FUNCTION_BLOCK RequestManager (* Basic Function Block Type *)
  (* Standard: 61499-2 *)
  (* Version 0.0, 9/24/2026, macie, Schneider Electric, Template *)
  PACKAGE Main;
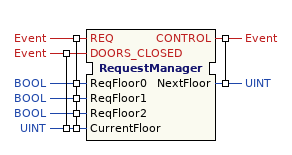
  EVENT_INPUT
    REQ WITH ReqFloor0, ReqFloor1, ReqFloor2, CurrentFloor; (* Normal Execution Request *)
    DOORS_CLOSED WITH CurrentFloor;
  END_EVENT
  EVENT_OUTPUT
    CONTROL WITH NextFloor; (* Initialization Confirm *)
  END_EVENT
  VAR_INPUT
    ReqFloor0 : BOOL;
    ReqFloor1 : BOOL;
    ReqFloor2 : BOOL;
    CurrentFloor : UINT;
  END_VAR
  VAR_OUTPUT
    NextFloor : UINT := 2; (* Output event qualifier *)
  END_VAR
  VAR
    Queue : ARRAY [0..2] OF UINT := [3(0)];
    MaxPriority : UINT;
    FloorPriority : UINT;
    QueueActive : BOOL := FALSE;
  END_VAR
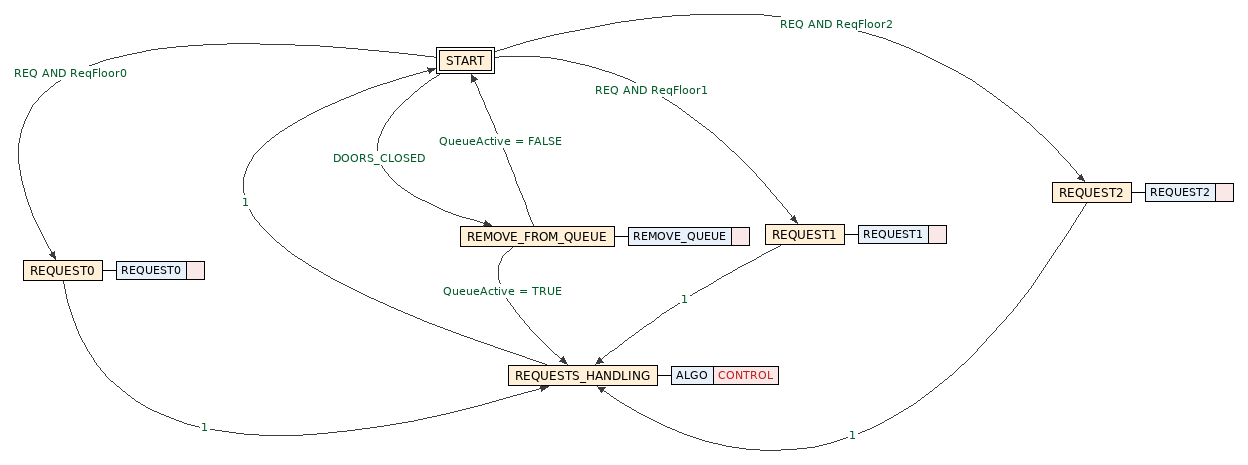
  EC_STATES
    START; (* Initial State *)
    REMOVE_FROM_QUEUE : REMOVE_QUEUE;
    REQUEST0 : REQUEST0;
    REQUEST1 : REQUEST1;
    REQUEST2 : REQUEST2;
    REQUESTS_HANDLING : ALGO -> CONTROL;
  END_STATES
  EC_TRANSITIONS
    START TO REMOVE_FROM_QUEUE := DOORS_CLOSED;
    START TO REQUEST0 := REQ AND ReqFloor0;
    REQUEST0 TO REQUESTS_HANDLING := 1;
    REQUEST1 TO REQUESTS_HANDLING := 1;
    REQUEST2 TO REQUESTS_HANDLING := 1;
    START TO REQUEST1 := REQ AND ReqFloor1;
    START TO REQUEST2 := REQ AND ReqFloor2;
    REMOVE_FROM_QUEUE TO START := QueueActive = FALSE;
    REMOVE_FROM_QUEUE TO REQUESTS_HANDLING := QueueActive = TRUE;
    REQUESTS_HANDLING TO START := 1;
  END_TRANSITIONS
  ALGORITHM ALGO IN ST: (* Initialization algorithm *)
;

NextFloor := CurrentFloor;
QueueActive := TRUE;
IF Queue[0] = 1 THEN
    IF CurrentFloor = 2 AND (Queue[1] > 0) THEN
        NextFloor := 1; (* Przystanek na 1 *)
    ELSE
        NextFloor := 0;
    END_IF;

ELSIF Queue[1] = 1 THEN
    NextFloor := 1;

ELSIF Queue[2] = 1 THEN
    IF CurrentFloor = 0 AND (Queue[1] > 0) THEN
        NextFloor := 1; (* Przystanek na 1 *)
    ELSE
        NextFloor := 2;
    END_IF;
END_IF;


(* --- 4. AKTUALIZACJA FLAGI AKTYWNOŚCI KOLEJKI --- *)
(* Ponownie przeliczamy priorytet, bo mógł zostać wyzerowany w Sekcji 2 *)
MaxPriority := MAX(Queue[0], MAX(Queue[1], Queue[2]));

IF FloorPriority = 0 THEN
    QueueActive := FALSE;
ELSE
    QueueActive := TRUE;
END_IF;
  END_ALGORITHM
  ALGORITHM REMOVE_QUEUE IN ST:
;
MaxPriority := MAX(Queue[0], MAX(Queue[1], Queue[2]));
IF MaxPriority > 0 THEN

	FloorPriority := Queue[CurrentFloor];
	Queue[CurrentFloor] := 0;


	IF Queue[0] > FloorPriority THEN Queue[0] := Queue[0] - 1; END_IF;
	IF Queue[1] > FloorPriority THEN Queue[1] := Queue[1] - 1; END_IF;
	IF Queue[2] > FloorPriority THEN Queue[2] := Queue[2] - 1; END_IF;
END_IF;

(*Updated value*)
MaxPriority := MAX(Queue[0], MAX(Queue[1], Queue[2]));

IF MaxPriority > 0 THEN
	QueueActive := TRUE;
ELSE
	QueueActive := FALSE;
END_IF;
  END_ALGORITHM
  ALGORITHM REQUEST0 IN ST:
;
MaxPriority := MAX(Queue[0], MAX(Queue[1], Queue[2]));

IF ReqFloor0 AND (Queue[0] = 0) THEN
    MaxPriority := MaxPriority + 1;
    Queue[0] := MaxPriority;
END_IF;
  END_ALGORITHM
  ALGORITHM REQUEST1 IN ST:
;
MaxPriority := MAX(Queue[0], MAX(Queue[1], Queue[2]));

IF ReqFloor1 AND (Queue[1] = 0) THEN
    MaxPriority := MaxPriority + 1;
    Queue[1] := MaxPriority;
END_IF;
  END_ALGORITHM
  ALGORITHM REQUEST2 IN ST:
;
MaxPriority := MAX(Queue[0], MAX(Queue[1], Queue[2]));

IF ReqFloor2 AND (Queue[2] = 0) THEN
    MaxPriority := MaxPriority + 1;
    Queue[2] := MaxPriority;
END_IF;
  END_ALGORITHM
END_FUNCTION_BLOCK
